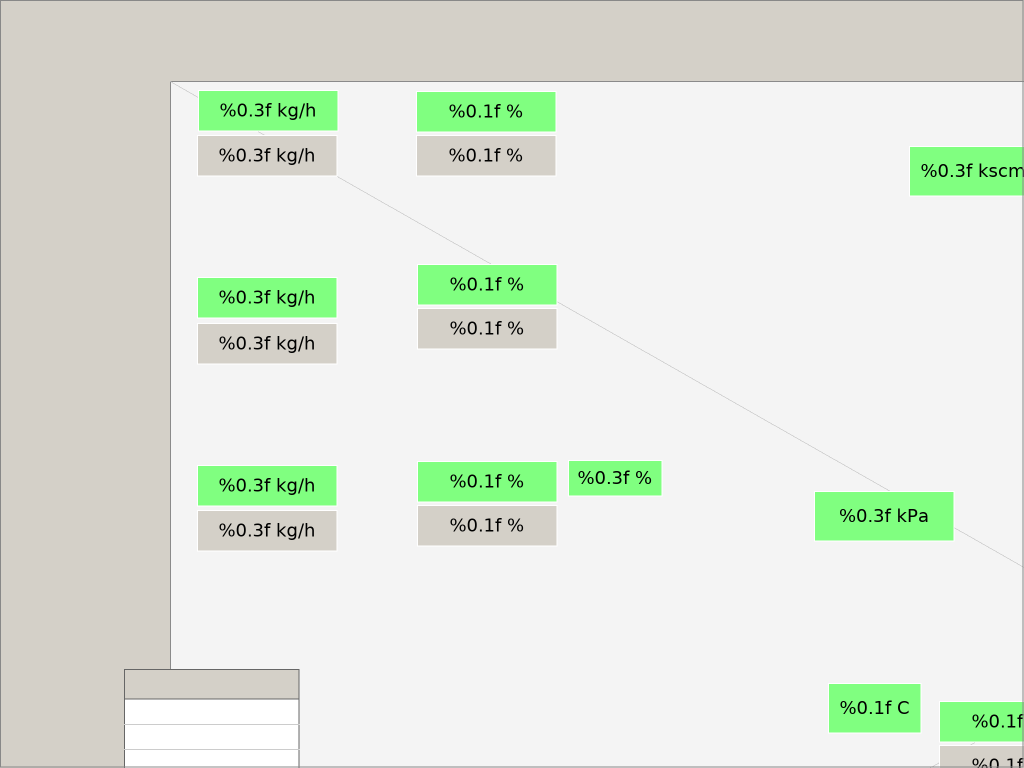
VISUALIZATION MainVisu  // 1024x768
    Image (170,81 1966x1119), image: ImagePool.base_diagram
    Rectangle (197,135 140x41), "%0.3f kg/h", text variable: G_IO.MBS_XMEAS[1]
    Rectangle (197,323 140x41), "%0.3f kg/h", text variable: G_IO.MBS_XMEAS[2]
    Rectangle (197,510 140x41), "%0.3f kg/h", text variable: G_IO.MBS_XMEAS[3]
    Rectangle (164,1031 140x50), "%0.3f kscmh", text variable: G_IO.XMEAS[4]
    Rectangle (909,146 140x50), "%0.3f kscmh", text variable: G_IO.XMEAS[5]
    Rectangle (492,858 140x50), "%0.3f kscmh", text variable: G_IO.XMEAS[6]
    Rectangle (814,491 140x50), "%0.3f kPa", text variable: G_IO.XMEAS[7]
    Rectangle (568,460 94x36), "%0.3f %", text variable: G_IO.XMEAS[8]
    Rectangle (671,890 92x50), "%0.1f C", text variable: G_IO.XMEAS[9]
    Rectangle (1941,152 140x50), "%0.3f kscmh", text variable: G_IO.XMEAS[10]
    Rectangle (1712,380 140x50), "%0.3f deg C", text variable: G_IO.XMEAS[11]
    Rectangle (1714,431 140x50), "%0.3f %", text variable: G_IO.XMEAS[12]
    Rectangle (1713,483 140x50), "%0.3f kPa", text variable: G_IO.XMEAS[13]
    Rectangle (1583,614 140x50), "%0.3f kPa", text variable: G_IO.XMEAS[14]
    Rectangle (1233,964 140x50), "%0.3f %", text variable: G_IO.XMEAS[15]
    Rectangle (1249,603 140x50), "%0.3f kPa", text variable: G_IO.XMEAS[16]
    Rectangle (1581,1157 140x50), "%0.3f cu. m/h", text variable: G_IO.XMEAS[17]
    Rectangle (1519,794 140x50), "%0.3f deg", text variable: G_IO.XMEAS[18]
    Rectangle (1439,296 140x50), "%0.3f kW", text variable: G_IO.XMEAS[20]
    Rectangle (828,683 93x50), "%0.1f C", text variable: G_IO.XMEAS[21]
    Rectangle (1180,273 140x50), "%0.3f deg C", text variable: G_IO.XMEAS[22]
    Table (2046,281 169x455), data array: VISU_MAIN.XMEAS_PurgeAnalyzer
        p3854506369: VISU_MAIN.XMEAS_PurgeAnalyzer[INDEX]
    Table (2049,809 169x283), data array: VISU_MAIN.XMEAS_ProductAnalyzer
        p3854506369: VISU_MAIN.XMEAS_ProductAnalyzer[INDEX]
    Table (124,669 175x334), data array: VISU_MAIN.XMEAS_FeedAnalyzer
        p3854506369: VISU_MAIN.XMEAS_FeedAnalyzer[INDEX]
    Rectangle (198,90 140x41), "%0.3f kg/h", text variable: G_IO.XMEAS[1]
    Rectangle (197,277 140x41), "%0.3f kg/h", text variable: G_IO.XMEAS[2]
    Rectangle (197,465 140x41), "%0.3f kg/h", text variable: G_IO.XMEAS[3]
    Rectangle (165,1085 140x41), "%0.3f kscmh", text variable: G_IO.MBS_XMEAS[4]
    Rectangle (416,91 140x41), "%0.1f %", text variable: G_IO.XMV[3]
    Rectangle (416,135 140x41), "%0.1f %", text variable: G_IO.NET_XMV[3]
    Rectangle (417,264 140x41), "%0.1f %", text variable: G_IO.XMV[2]
    Rectangle (417,308 140x41), "%0.1f %", text variable: G_IO.NET_XMV[2]
    Rectangle (417,461 140x41), "%0.1f %", text variable: G_IO.XMV[3]
    Rectangle (417,505 140x41), "%0.1f %", text variable: G_IO.NET_XMV[3]
    Rectangle (386,1157 101x41), "%0.1f %", text variable: G_IO.XMV[4]
    Rectangle (939,701 140x41), "%0.1f %", text variable: G_IO.XMV[10]
    Rectangle (939,745 140x41), "%0.1f %", text variable: G_IO.NET_XMV[4]
END_VISUALIZATION

(* stored: Version 1.1.0.1, ProductVersion 3.1.0.36
   Visu MainVisu: Id {e8b20c2b-5c8d-4eb0-9209-1744dfeeea02} *)
